FUNCTION_BLOCK FB_MUX_STRING (* See FB_MUX_ANY *)
  (* Standard: IEC 61499 *)
  (* Version 0.0, 2006-09-13, JHC, Holobloc Inc, Derived from FB_MUX_WSTRING. *)
  (* Compiler header: package fb.rt.strings; *)
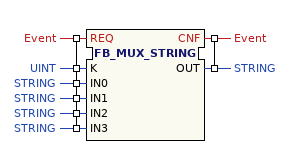
  EVENT_INPUT
    REQ WITH K, IN0, IN1, IN2, IN3;
  END_EVENT
  EVENT_OUTPUT
    CNF WITH OUT;
  END_EVENT
  VAR_INPUT
    K : UINT;
    IN0 : STRING;
    IN1 : STRING;
    IN2 : STRING;
    IN3 : STRING;
  END_VAR
  VAR_OUTPUT
    OUT : STRING;
  END_VAR
END_FUNCTION_BLOCK
